(* Logix 5000 project; controller testing vendor 1 type 14 code 151 rev 32.11; software revision 32.00 *)

TASK MainTask (continuous, watchdog 500 ms) : MainProgram

MODULES
   Local : vendor 1 type 14 code 151 (Compact 0, rev 32.11)
      Analog_IO : Embedded (Compact 2, rev 1.1, Output RPI 80 ms)
      Counters : Embedded (Compact 3, rev 1.1, Output RPI 20 ms)
      Discrete_IO : Embedded (Compact 1, rev 3.1, Output RPI 20 ms)
END_MODULES

TYPE test :
STRUCT
   value1 : DINT;
   value2 : STRING;
   value3 : INT;
   value4 : BOOL;
   value5 : DINT[5];
END_STRUCT
END_TYPE

VAR_GLOBAL   (* controller tags *)
   counttest : COUNTER := (PRE := 9999, ACC := 4232);
   DataReadfromPLC : BOOL;
   DataReadPLC : DINT[10] := ([0] := 245, [1] := 3633, [2] := 7777, [3] := 356636, [4] := 346363, [5] := 99999, [6] := 3843, [7] := 9990, [8] := 4111);
   DataSend : BOOL := 1;
   Dummy : BOOL := 1;
   Gotackfromplc : BOOL;
   KeepTimer : TIMER := (PRE := 3500, ACC := 287, EN := 1, TT := 1);
   Mach_Auto : BOOL := 1;
   moreTags1 : DINT;
   moretags2 : DINT;
   moretags3 : DINT;
   moretags4 : DINT;
   moretags5 : DINT;
   Movenum : DINT;
   movenumctr : COUNTER := (PRE := 99999, ACC := 819);
   movenumtimer : TIMER := (PRE := 2500, ACC := 1667, EN := 1, TT := 1);
   ons_this : BOOL;
   reset : TIMER := (PRE := 500);
   string1 : STRING := 'testing1';
   string2 : STRING := 'testing2';
   string3 : STRING := 'testing3';
   string4 : STRING := 'testing4';
   string5 : STRING := 'testing5';
   string6 : STRING := 'testing6';
   string7 : STRING := '819';
   string8 : STRING := '4yere';
   string9 : STRING := 'dgdgdg';
   string_array : STRING[10] := ([0] := 'testing2', [1] := 'testing3', [2] := 'testing4', [3] := 'testing5', [4] := 'testing6', [5] := '819', [6] := '4yere', [7] := 'dgdgdg');
   stringread : STRING := 'testing1';
   test_array : DINT[5] := ([0] := 345, [1] := 5665, [2] := 456, [3] := 113121, [4] := 121314);
   udt_Item : test := (value1 := 367, value2 := 'testing2', value3 := 4232, value4 := 1, value5[0] := 5000, value5[1] := 923);
END_VAR

PROGRAM MainProgram   (* main routine MainRoutine *)
VAR
   Send_data : BOOL := 1;
END_VAR

ROUTINE MainRoutine   (* ladder *)
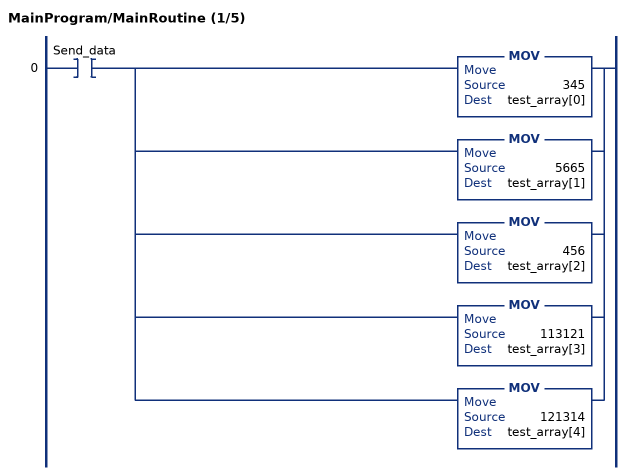
   0: XIC(Send_data)[MOV(345,test_array[0]) ,MOV(5665,test_array[1]) ,MOV(456,test_array[2]) ,MOV(113121,test_array[3]) ,MOV(121314,test_array[4]) ];
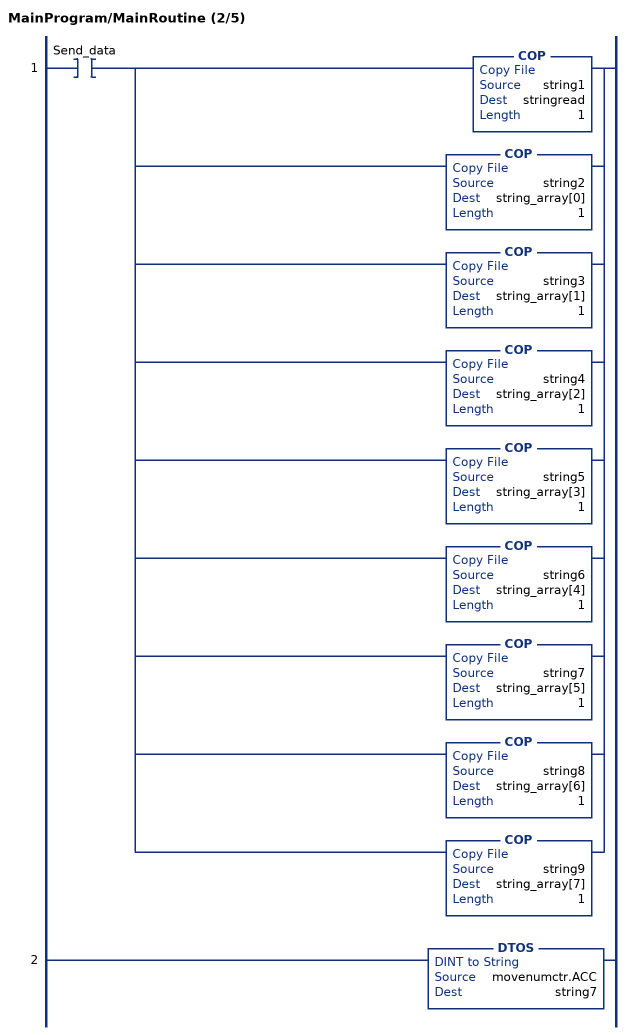
   1: XIC(Send_data)[COP(string1,stringread,1) ,COP(string2,string_array[0],1) ,COP(string3,string_array[1],1) ,COP(string4,string_array[2],1) ,COP(string5,string_array[3],1) ,COP(string6,string_array[4],1) ,COP(string7,string_array[5],1) ,COP(string8,string_array[6],1) ,COP(string9,string_array[7],1) ];
   2: DTOS(movenumctr.ACC,string7);
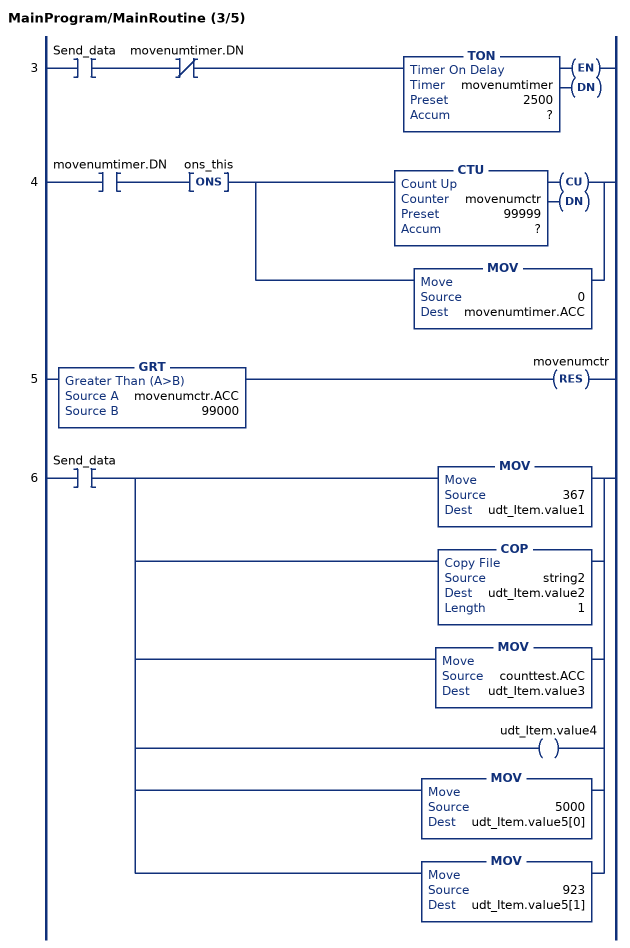
   3: XIC(Send_data)XIO(movenumtimer.DN)TON(movenumtimer,?,?);
   4: XIC(movenumtimer.DN)ONS(ons_this)[CTU(movenumctr,?,?) ,MOV(0,movenumtimer.ACC) ];
   5: GRT(movenumctr.ACC,99000)RES(movenumctr);
   6: XIC(Send_data)[MOV(367,udt_Item.value1) ,COP(string2,udt_Item.value2,1) ,MOV(counttest.ACC,udt_Item.value3) ,OTE(udt_Item.value4) ,MOV(5000,udt_Item.value5[0]) ,MOV(923,udt_Item.value5[1]) ];
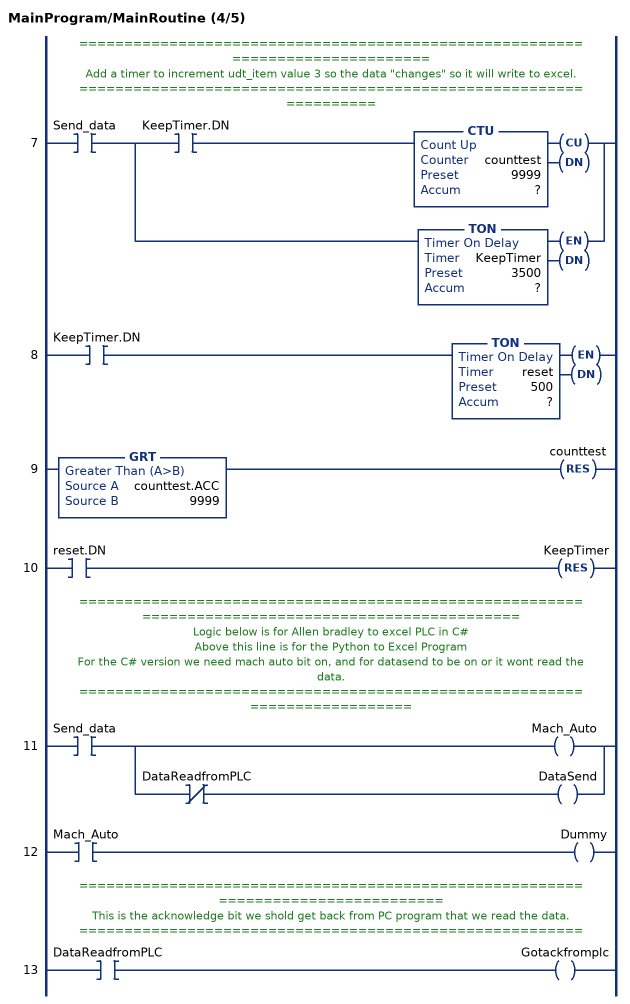
   // ==============================================================================
   // Add a timer to increment udt_item value 3 so the data "changes" so it will write to excel.
   // ==================================================================
   7: XIC(Send_data)[XIC(KeepTimer.DN) CTU(counttest,?,?) ,TON(KeepTimer,?,?) ];
   8: XIC(KeepTimer.DN)TON(reset,?,?);
   9: GRT(counttest.ACC,9999)RES(counttest);
   10: XIC(reset.DN)RES(KeepTimer);
   // ==================================================================================================
   // Logic below is for Allen bradley to excel PLC in C#
   // Above this line is for the Python to Excel Program
   // For the C# version we need mach auto bit on, and for datasend to be on or it wont read the data.
   // ==========================================================================
   11: XIC(Send_data)[OTE(Mach_Auto) ,XIO(DataReadfromPLC) OTE(DataSend) ];
   12: XIC(Mach_Auto)OTE(Dummy);
   // =================================================================================
   // This is the acknowledge bit we shold get back from PC program that we read the data.
   // ========================================================
   13: XIC(DataReadfromPLC)OTE(Gotackfromplc);
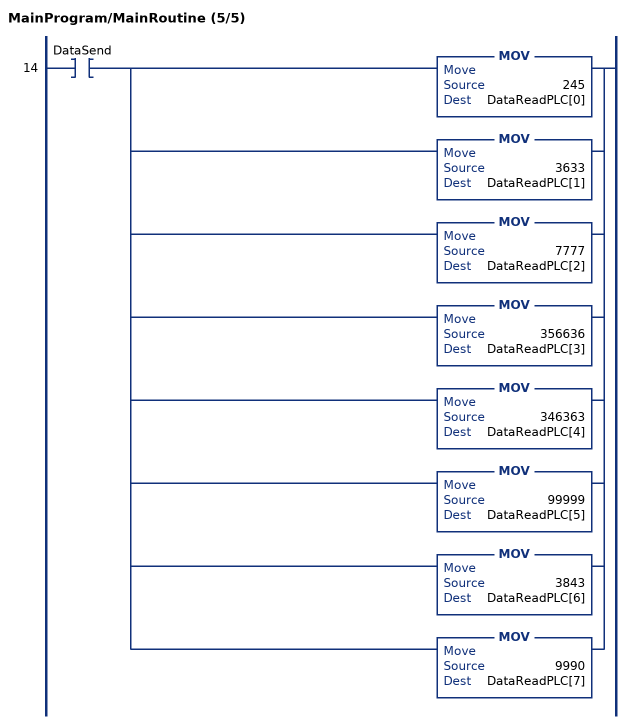
   14: XIC(DataSend)[MOV(245,DataReadPLC[0]) ,MOV(3633,DataReadPLC[1]) ,MOV(7777,DataReadPLC[2]) ,MOV(356636,DataReadPLC[3]) ,MOV(346363,DataReadPLC[4]) ,MOV(99999,DataReadPLC[5]) ,MOV(3843,DataReadPLC[6]) ,MOV(9990,DataReadPLC[7]) ];
END_ROUTINE
END_PROGRAM
